TYPE IoSh10pilShutter :
STRUCT
	InputMagneticSwitch1	AT %I* : BOOL;	
	InputMagneticSwitch2	AT %I* : BOOL;		
	OutputSwitchContactClosure	AT %Q* : BOOL;	
END_STRUCT
END_TYPE

(* stored: Version 1.1.0.1, ProductVersion 3.1.4024.4
   DUT IoSh10pilShutter: Id {ac387f79-a4ea-4d0c-ac0a-72c25e0679fb} *)
